FUNCTION_BLOCK SystemControl
VAR_IN_OUT
	motor_axis : Tc2_MC2.AXIS_REF;
	system_control_param : SystemControlParam;
	motor_state : MotorState;
END_VAR
VAR_OUTPUT
	target_velocity : LREAL;
END_VAR
VAR
	motorPower : Tc2_MC2.MC_Power;
END_VAR

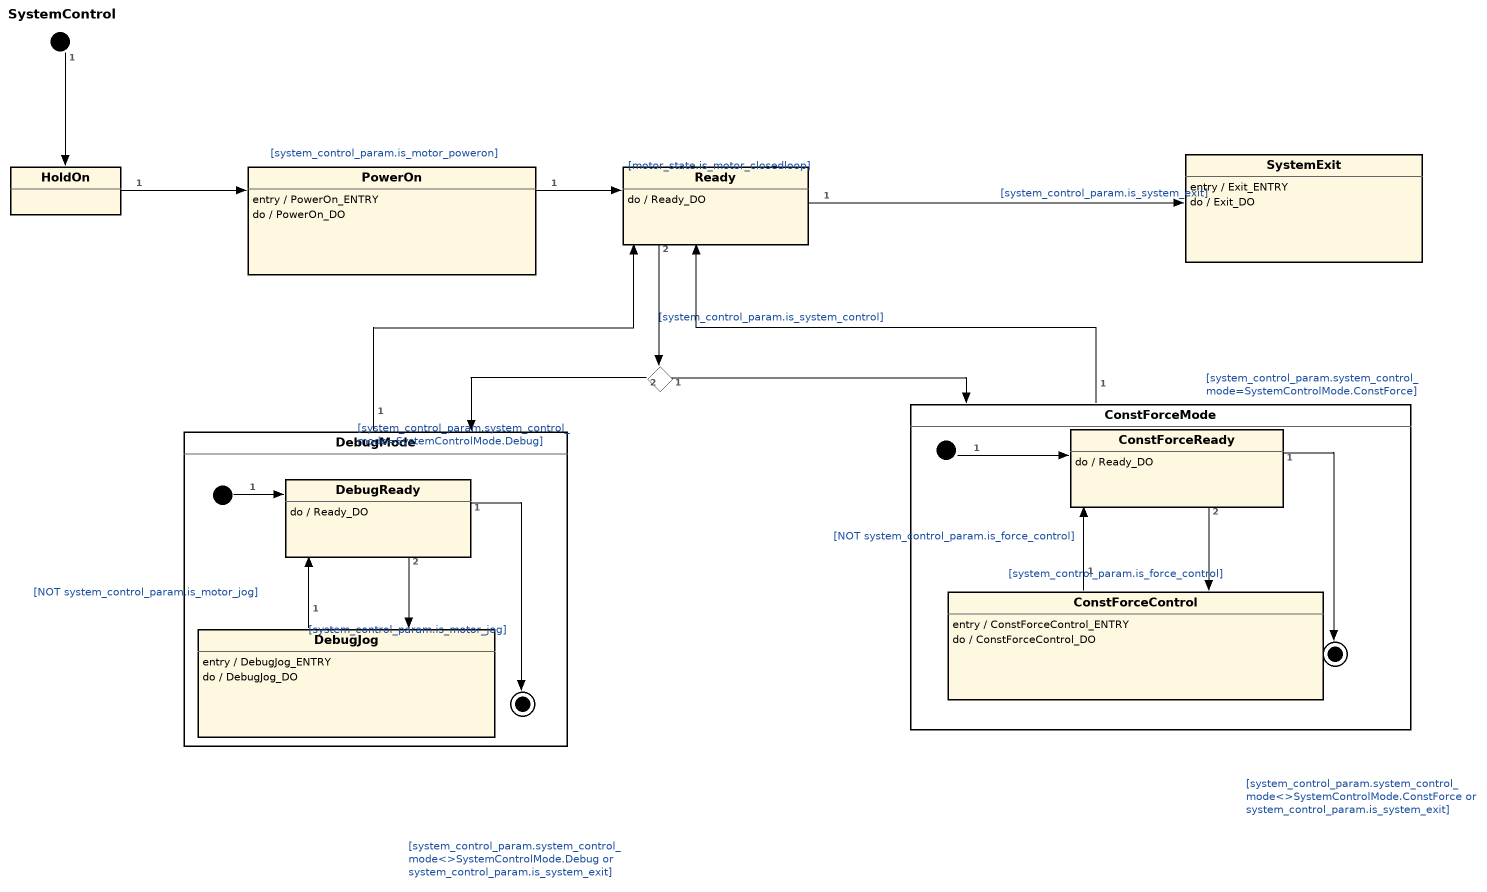
STATECHART SystemControl  // abortable
    START StartState1
    STATE HoldOn
    STATE PowerOn
        entry / PowerOn_ENTRY
        do / PowerOn_DO
    STATE Ready
        do / Ready_DO
    STATE SystemExit
        entry / Exit_ENTRY
        do / Exit_DO
    CHOICE ChoiceElement1
    COMPOSITE STATE ConstForceMode
        START StartState3
        STATE ConstForceReady
            do / Ready_DO
        STATE ConstForceControl
            entry / ConstForceControl_ENTRY
            do / ConstForceControl_DO
        END EndState2
        StartState3 -> ConstForceReady  // priority 1, on completion
        ConstForceReady -> EndState2 [system_control_param.system_control_mode<>SystemControlMode.ConstForce or system_control_param.is_system_exit] // priority 1
        ConstForceReady -> ConstForceControl [system_control_param.is_force_control] // priority 2
        ConstForceControl -> ConstForceReady [NOT system_control_param.is_force_control] // priority 1
    END_STATE
    COMPOSITE STATE DebugMode
        START StartState2
        STATE DebugReady
            do / Ready_DO
        STATE DebugJog
            entry / DebugJog_ENTRY
            do / DebugJog_DO
        END EndState1
        StartState2 -> DebugReady  // priority 1, on completion
        DebugReady -> EndState1 [system_control_param.system_control_mode<>SystemControlMode.Debug or system_control_param.is_system_exit] // priority 1
        DebugReady -> DebugJog [system_control_param.is_motor_jog] // priority 2
        DebugJog -> DebugReady [NOT system_control_param.is_motor_jog] // priority 1
    END_STATE
    StartState1 -> HoldOn  // priority 1, on completion
    HoldOn -> PowerOn [system_control_param.is_motor_poweron] // priority 1
    PowerOn -> Ready [motor_state.is_motor_closedloop] // priority 1
    Ready -> SystemExit [system_control_param.is_system_exit] // priority 1
    Ready -> ChoiceElement1 [system_control_param.is_system_control] // priority 2
    ChoiceElement1 -> ConstForceMode [system_control_param.system_control_mode=SystemControlMode.ConstForce] // priority 1
    ChoiceElement1 -> DebugMode [system_control_param.system_control_mode=SystemControlMode.Debug] // priority 2
    ConstForceMode -> Ready  // priority 1, on completion
    DebugMode -> Ready  // priority 1, on completion
END_STATECHART

ACTION ConstForceControl_DO:

END_ACTION

ACTION ConstForceControl_ENTRY:

END_ACTION

ACTION DebugJog_DO:
target_velocity := system_control_param.jog_param.jog_velocity;
END_ACTION

ACTION DebugJog_ENTRY:

END_ACTION

ACTION Exit_DO:
motorPower(
	Axis:= motor_axis, 
	Enable:= FALSE, 
	Enable_Positive:= TRUE, 
	Enable_Negative:= TRUE, 
	Override:= , 
	BufferMode:= , 
	Options:= , 
	Status=> , 
	Busy=> , 
	Active=> , 
	Error=> , 
	ErrorID=> );
END_ACTION

ACTION Exit_ENTRY:
target_velocity := 0;
END_ACTION

ACTION PowerOn_DO:
motorPower(
	Axis:= motor_axis, 
	Enable:= TRUE, 
	Enable_Positive:= TRUE, 
	Enable_Negative:= TRUE, 
	Override:= , 
	BufferMode:= , 
	Options:= , 
	Status=> , 
	Busy=> , 
	Active=> , 
	Error=> , 
	ErrorID=> );
END_ACTION

ACTION PowerOn_ENTRY:

END_ACTION

ACTION Ready_DO:
target_velocity := 0;
END_ACTION

END_FUNCTION_BLOCK

(* stored: Version 1.1.0.1, ProductVersion 3.1.4024.11
   POU SystemControl: Id {f26ced33-dea7-45dd-a280-164c04479403}, SpecialFunc None
   Action ConstForceControl_DO: Id {5eebccd2-8522-43d7-816e-067ac0802640}
   Action ConstForceControl_ENTRY: Id {8357e1b7-88f6-41cf-bfa0-7aeebec320b9}
   Action DebugJog_DO: Id {8c36f437-5ca7-417b-b37b-159c749d264e}
   Action DebugJog_ENTRY: Id {535b0c77-eda4-474a-9745-c61a2f1cf3e4}
   Action Exit_DO: Id {958c05c9-7223-4cd3-ae6c-85dda310b19b}
   Action Exit_ENTRY: Id {e0dc1617-e455-45fd-94e8-27be8ae21ef5}
   Action PowerOn_DO: Id {949cde52-772c-440d-8e0a-69f5e6463c55}
   Action PowerOn_ENTRY: Id {3acfe3ac-6e8d-41f2-8066-0b7dd094679c}
   Action Ready_DO: Id {4707b248-c668-4be3-ae90-41598c95ecf2} *)
